TYPE U_GEAR_DATA :
UNION
  stData              : ARRAY[1..MAX_MOVER] OF ST_GEAR_DATA;

  byData    AT %Q*    : ARRAY[1..MAX_MOVER] OF
                        ARRAY[1..SIZEOF(ST_GEAR_DATA)] OF BYTE;
END_UNION
END_TYPE

(* stored: Version 1.1.0.1
   DUT U_GEAR_DATA: Id {222697a6-e0c0-42fd-bc8e-7d82a4ad4a08} *)
